PROGRAM MAIN
VAR
END_VAR


// Call Programs
PRG1_Conveyer_Operation();
PRG2_Object_Detection();

END_PROGRAM

(* stored: Version 1.1.0.1, ProductVersion 3.1.4024.12
   POU MAIN: Id {39088c10-7eec-42b3-bfb0-956326d32e9e}, SpecialFunc None *)
